TYPE ST_ACSwitchgear_Get :
STRUCT
	b_InputSectionAvailable	: BOOL;
	b_InputMCCBfb			: BOOL;
	b_InputMCCBShuntOK		: BOOL;	
	b_OutputMCCBfb			: BOOL;
	b_OutputMCCBShuntOK		: BOOL;
	b_CEEprefuseOK			: BOOL;
	b_InputSynchronizerfb	: BOOL;
	b_InputContactorfb		: BOOL;
	b_PENlinkfb				: BOOL;
	events					: ST_ACswitchgear_events;
END_STRUCT
END_TYPE

(* stored: Version 1.1.0.1, ProductVersion 3.1.4026.18
   DUT ST_ACSwitchgear_Get: Id {fd35a08c-e6a5-4d67-ac0a-fbbc559fc1ed} *)
